FUNCTION_BLOCK FB_Descargadro_SFC
VAR_INPUT
	//nuestras_variables
	pieza_ok: BOOL;	

    // SFC-Flags
    SFCPause: BOOL;
    SFCReset: BOOL;
    
    // Indicadores de sincronizacion
    Ack: BOOL := TRUE;
    Execute: BOOL;
	
	//Entradas
    Horizontal_descargador_detras: BOOL;
	Vertical_descargador_abajo: BOOL;
	Vacio_obtenido_vacuostato_descargador: BOOL;
	Vertical_descargador_arriba: BOOL;
	Horizontal_descargador_delante: BOOL;
	Vertical_descargador_arriba: BOOL;
	
END_VAR
VAR_OUTPUT
    // Indicadores de sincronizacion
    Done: BOOL;
    Ready: BOOL;

	//Salidas
	Descargador_atras: BOOL;
END_VAR
VAR
END_VAR

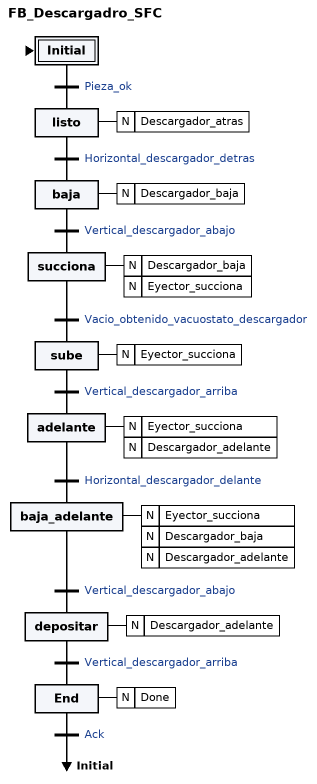
INITIAL_STEP Initial:
END_STEP
TRANSITION FROM Initial TO listo
    := Pieza_ok;
END_TRANSITION
STEP listo:
    Descargador_atras(N);
END_STEP
TRANSITION FROM listo TO baja
    := Horizontal_descargador_detras;
END_TRANSITION
STEP baja:
    Descargador_baja(N);
END_STEP
TRANSITION FROM baja TO succiona
    := Vertical_descargador_abajo;
END_TRANSITION
STEP succiona:
    Descargador_baja(N);
    Eyector_succiona(N);
END_STEP
TRANSITION FROM succiona TO sube
    := Vacio_obtenido_vacuostato_descargador;
END_TRANSITION
STEP sube:
    Eyector_succiona(N);
END_STEP
TRANSITION FROM sube TO adelante
    := Vertical_descargador_arriba;
END_TRANSITION
STEP adelante:
    Eyector_succiona(N);
    Descargador_adelante(N);
END_STEP
TRANSITION FROM adelante TO baja_adelante
    := Horizontal_descargador_delante;
END_TRANSITION
STEP baja_adelante:
    Eyector_succiona(N);
    Descargador_baja(N);
    Descargador_adelante(N);
END_STEP
TRANSITION FROM baja_adelante TO depositar
    := Vertical_descargador_abajo;
END_TRANSITION
STEP depositar:
    Descargador_adelante(N);
END_STEP
TRANSITION FROM depositar TO End
    := Vertical_descargador_arriba;
END_TRANSITION
STEP End:
    Done(N);
END_STEP
TRANSITION FROM End TO Initial
    := Ack;
END_TRANSITION

END_FUNCTION_BLOCK

(* stored: Version 1.1.0.1, ProductVersion 3.1.4024.12
   POU FB_Descargadro_SFC: Id {f35099df-5230-41a2-ba70-222d8682b89d}, SpecialFunc None *)
